TYPE ST_System_MVWW_Stellwert :
STRUCT
	Anford_Stellventil		: BOOL;
	Anford_Pumpe			: BOOL;
	Einschaltperiode_Max	: TIME := T#5S;
	Einschalten				: BOOL;
	Modus_Pumpe				: SINT;
	Sollw_Pumpe				: REAL;
END_STRUCT
END_TYPE

(* stored: Version 1.1.0.1, ProductVersion 3.1.4024.9
   DUT ST_System_MVWW_Stellwert: Id {c305e3f1-9058-4035-952f-abbe3c8d507f} *)
